% RSLogix 500 project P1 - Digital Control Logic.RSS, saved by version 8.30.00.16 %
PROJECT "PROJECT1"    % processor: Bul.1763 MicroLogix 1100 Series B %

PROGRAM FILES
  LAD 2 "MAIN"  4 rungs
  LAD 3 "IO"  5 rungs
  LAD 4 "CONTROLS"  5 rungs
  LAD 5 "ALARMS"  1 rungs

DATA FILES
  O0 OUTPUT  7 elements
  I1 INPUT  12 elements
  S2 STATUS  66 elements
  B3 BINARY  1 elements
  T4 TIMER  2 elements
  C5 COUNTER  1 elements
  R6 CONTROL  1 elements
  N7 INTEGER  1 elements
  F8 FLOAT  1 elements

LADDER 2 "MAIN"
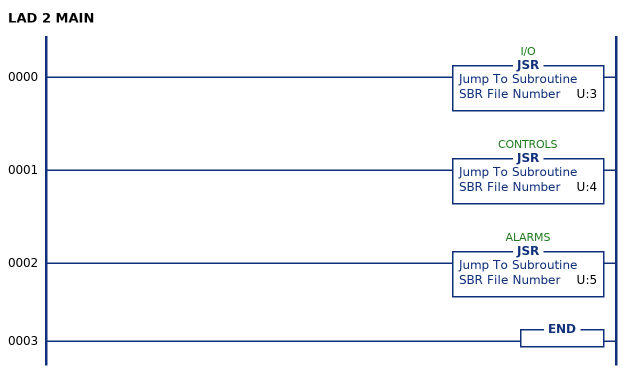
% Rung: 0 %
SOR JSR U:3 EOR
%   U:3  "I/O" %
% Rung: 1 %
SOR JSR U:4 EOR
%   U:4  "CONTROLS" %
% Rung: 2 %
SOR JSR U:5 EOR
%   U:5  "ALARMS" %
% Rung: 3 %
SOR END EOR

LADDER 3 "IO"
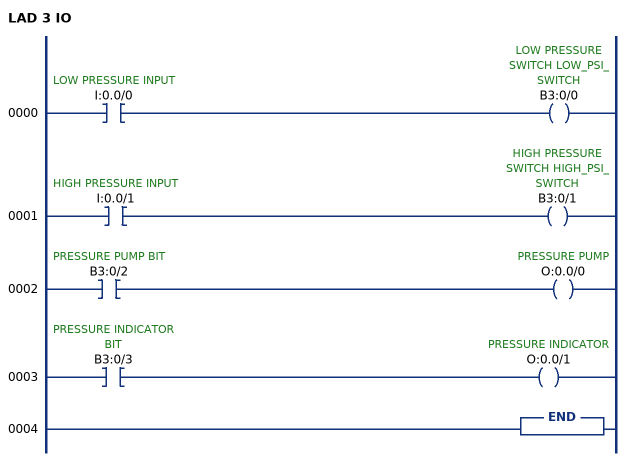
% Rung: 0 %
SOR XIC I:0.0/0 OTE B3:0/0 EOR
%   I:0.0/0  "LOW PRESSURE INPUT" %
%   B3:0/0  LOW_PSI_SWITCH  "LOW PRESSURE SWITCH" %
% Rung: 1 %
SOR XIC I:0.0/1 OTE B3:0/1 EOR
%   I:0.0/1  "HIGH PRESSURE INPUT" %
%   B3:0/1  HIGH_PSI_SWITCH  "HIGH PRESSURE SWITCH" %
% Rung: 2 %
SOR XIC B3:0/2 OTE O:0.0/0 EOR
%   B3:0/2  "PRESSURE PUMP BIT" %
%   O:0.0/0  "PRESSURE PUMP" %
% Rung: 3 %
SOR XIC B3:0/3 OTE O:0.0/1 EOR
%   B3:0/3  "PRESSURE INDICATOR BIT" %
%   O:0.0/1  "PRESSURE INDICATOR" %
% Rung: 4 %
SOR END EOR

LADDER 4 "CONTROLS"
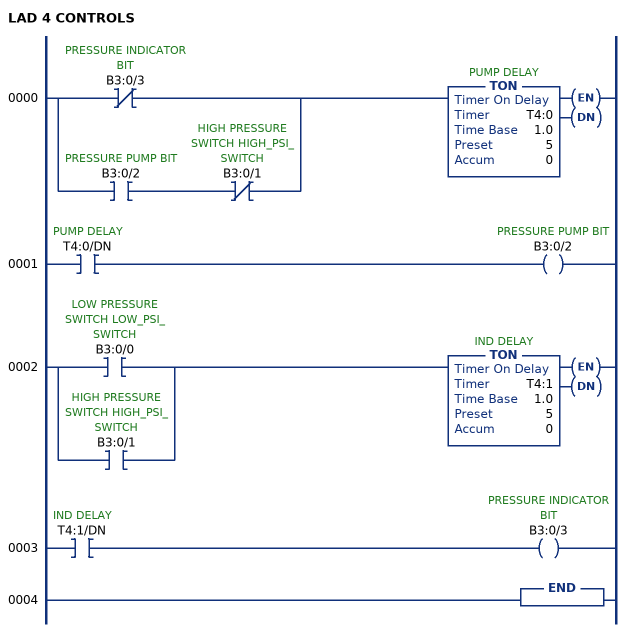
% Rung: 0 %
SOR BST XIO B3:0/3 NXB XIC B3:0/2 XIO B3:0/1 BND TON T4:0 1.0 5 0 EOR
%   B3:0/3  "PRESSURE INDICATOR BIT" %
%   B3:0/2  "PRESSURE PUMP BIT" %
%   B3:0/1  HIGH_PSI_SWITCH  "HIGH PRESSURE SWITCH" %
%   T4:0  "PUMP DELAY" %
% Rung: 1 %
SOR XIC T4:0/DN OTE B3:0/2 EOR
%   T4:0  "PUMP DELAY" %
%   B3:0/2  "PRESSURE PUMP BIT" %
% Rung: 2 %
SOR BST XIC B3:0/0 NXB XIC B3:0/1 BND TON T4:1 1.0 5 0 EOR
%   B3:0/0  LOW_PSI_SWITCH  "LOW PRESSURE SWITCH" %
%   B3:0/1  HIGH_PSI_SWITCH  "HIGH PRESSURE SWITCH" %
%   T4:1  "IND DELAY" %
% Rung: 3 %
SOR XIC T4:1/DN OTE B3:0/3 EOR
%   T4:1  "IND DELAY" %
%   B3:0/3  "PRESSURE INDICATOR BIT" %
% Rung: 4 %
SOR END EOR

OTHER DOCUMENTED ADDRESSES
  B3:0/4  "ONE SHOT PUMP"
  B3:0/5  "ONE SHOT PUMP"
  B3:1/0  "PRESSURE INCREASE TRIGGER BIT"
  B30:0/0  "LOW PRESSURE SWITCH BIT"
  I:0  "LOW PRESSURE SWITCH"
  I:1  "HIGH PRESSURE SWITCH"
  O:0  "Pressure Pump"
  O:1  PRESSURE_INDICATOR  "PRESSURE INDICATOR LIGHT"

DATA TABLE (non-zero values as saved)
DATA T4
% .PRE .ACC %
% T4:0 % 5 0
% T4:1 % 5 0
